(* PLC project mbNewproject.project, Prosoft-Systems Ltd. Astra.IDE Astra.IDE V1.7.0.0 *)
(* stored: creationDateTime 2023-08-18T10:12:58.0723218, modificationDateTime 2023-08-17T12:00:25.8272152 *)
